PROGRAM sub_Measure
VAR
		fbWaterConsumption			:	FB_Count;
		fbWaterConsumptionZisterne	:	FB_Count;
		
		fbHumWohnzimmer		:	FB_Convert_10V2relHum;
		fbHumTechnikraum	:	FB_Convert_10V2relHum;
		fbHumWerkstatt		:	FB_Convert_10V2relHum;
		fbHumGarage			:	FB_Convert_10V2relHum;
		
		fbCO2Wohnzimmer		:	FB_Convert_10V2co2;
		
		fbZisterne			:	FB_Convert_mA2Zisterne;
		
		fbTempGarage		:	FB_Convert_10V2temp;
		fbTempWerkstatt		:	FB_Convert_10V2temp;
		fbTempTechnikraum	:	FB_Convert_10V2temp;
		fbTempWohnzimmer	:	FB_Convert_10V2temp;
END_VAR

//###################################################################################
//##-----------------------------------MEASUREMENT---------------------------------##
//###################################################################################


gvl_mb.Output_Registers[19] := INT_TO_WORD(gvl_EA.iIAPT_01_1);	// Temperatur Bühne

//--------------------WATER CONSUMPTION Trinkwasser (1 = 10 Liter)-------------------
fbWaterConsumption
(
	bInput			:= gvl_EA.bID24_03_3,
	bAllFlanks 		:= FALSE,
	wCountRetain	:= gvl_RETAIN.waterConsumption,
	wOut			=> gvl_mb.Output_Registers[0]
);
//-----------------------------------------------------------------------
//--------------------WATER CONSUMPTION Zisterne (1 = 1 Liter)-------------------
fbWaterConsumptionZisterne
(
	bInput			:= gvl_EA.bID24_03_4,
	bAllFlanks 		:= FALSE,
	wCountRetain	:= gvl_RETAIN.waterConsumptionZisterne,
	wOut			=> gvl_mb.Output_Registers[22]
);
//-----------------------------------------------------------------------
//--------------------HUMIDITY WOHNZIMMER--------------------------------
fbHumWohnzimmer
(
	iInput		:= gvl_EA.iIAV01_2,
	tRefresh 	:= T#10S,
	wOut 		=> gvl_mb.Output_Registers[15]
);
//-----------------------------------------------------------------------
//--------------------HUMIDITY TECHNIKRAUM--------------------------------
fbHumTechnikraum
(
	iInput		:= gvl_EA.iIAV02_1,
	tRefresh 	:= T#10S,
	wOut 		=> gvl_mb.Output_Registers[18]
);
//-----------------------------------------------------------------------
//--------------------HUMIDITY WERKSTATT--------------------------------
fbHumWerkstatt
(
	iInput		:= gvl_EA.iWIAV01_2,
	tRefresh 	:= T#10S,
	wOut 		=> gvl_mb.Output_Registers[21]
);
//-----------------------------------------------------------------------
//--------------------HUMIDITY GARAGE--------------------------------
fbHumGarage
(
	iInput		:= gvl_EA.iWIAV01_3,
	tRefresh 	:= T#10S,
	wOut 		=> gvl_mb.Output_Registers[24]
);
//-----------------------------------------------------------------------
//--------------------CO2 WOHNZIMMER-------------------------------------
fbCO2Wohnzimmer
(
	iInput		:= gvl_EA.iIAV01_3,
	tRefresh 	:= T#10S,
	wOut 		=> gvl_mb.Output_Registers[16]
);
//-----------------------------------------------------------------------
//--------------------TEMP GARAGE-------------------------------------
fbTempGarage
(
	iInput		:= gvl_EA.iWIAV01_4,
	tRefresh 	:= T#10S,
	itempMAX	:= 70,
	itempMIN	:= -30,
	wOut 		=> gvl_mb.Output_Registers[23]
);
//-----------------------------------------------------------------------
//--------------------TEMP WERKSTATT-------------------------------------
fbTempWerkstatt
(
	iInput		:= gvl_EA.iWIAV01_1,
	tRefresh 	:= T#10S,
	itempMAX	:= 70,
	itempMIN	:= -30,
	wOut 		=> gvl_mb.Output_Registers[20]
);
//-----------------------------------------------------------------------
//--------------------TEMP TECHNIKRAUM-------------------------------------
fbTempTechnikraum
(
	iInput		:= gvl_EA.iIAV01_4,
	tRefresh 	:= T#10S,
	itempMAX	:= 70,
	itempMIN	:= -30,
	wOut 		=> gvl_mb.Output_Registers[17]
);
//-----------------------------------------------------------------------
//--------------------TEMP WOHNZIMMER-------------------------------------
fbTempWohnzimmer
(
	iInput		:= gvl_EA.iIAV01_1,
	tRefresh 	:= T#10S,
	itempMAX	:= 50,
	itempMIN	:= 0,
	wOut 		=> gvl_mb.Output_Registers[14]
);
//-----------------------------------------------------------------------
//--------------------ZISTERNE-------------------------------------
fbZisterne
(
	iInput		:= gvl_EA.iIAA01_1,
	tRefresh 	:= T#1M,
	wOutPerc	=> gvl_mb.Output_Registers[12],
	wOutLiter	=> gvl_mb.Output_Registers[13]

);
//-----------------------------------------------------------------------

END_PROGRAM

(* stored: Version 1.1.0.1, ProductVersion 3.1.4024.4
   POU sub_Measure: Id {c86e02d1-7a17-45fa-8e50-215beceed17d}, SpecialFunc None *)
